{attribute 'qualified_only'}
VAR_GLOBAL
	t_global	:	REAL;
	t_cycle		:	REAL;
END_VAR

(* stored: Version 1.1.0.1, ProductVersion 3.1.4022.12
   GVL GVL: Id {939af1df-f911-4151-89bf-60df41444175} *)
